INTERFACE I_AveNadadora

END_INTERFACE

(* stored: Version 1.1.0.1, ProductVersion 3.1.4024.12
   Itf I_AveNadadora: Id {599ea192-3695-4ff2-97e1-c2a8a2bf0546} *)
